(* IEC 61131-3 sources: AXOpen/src/showcase/app/src/components.dukane.welders/Documentation, 3 files *)

(* ---- Axo_IQ_SeriesWelder_Showcase.st ---- *)
USING AXOpen.Core;
NAMESPACE AXOpen.Components.Dukane.Welders
    {S7.extern=ReadWrite}
    CLASS Axo_IQ_SeriesWelder_Showcase EXTENDS AXOpen.Core.AxoObject
        //<ComponentDeclaration>
        VAR PUBLIC
            Dukane_IQ_SeriesWelder : AXOpen.Components.Dukane.Welders.Axo_IQ_SeriesWelder;
        END_VAR
        //</ComponentDeclaration>

        //<InitializationArgumentsDeclaration>
        VAR PUBLIC
            {#ix-set:AttributeName = "<#Activate manual control#>"}
            ActivateManualControl : BOOL;
        END_VAR
        //</InitializationArgumentsDeclaration>

        METHOD PUBLIC OVERRIDE Run
            VAR_INPUT
                inParent : IAxoObject;
            END_VAR

            SUPER.Run(inParent);

            IF ActivateManualControl THEN
                Dukane_IQ_SeriesWelder.ActivateManualControl();
            END_IF;

            //<Initialization>
            Dukane_IQ_SeriesWelder.Run(inParent := THIS, hwID := AXOpen.Showcase.HwIdentifiers#dukaneiqauto_HwID);
            //</Initialization>

        THIS.UseInSequencer();
        END_METHOD

        //<Usage>
        VAR PUBLIC
            {#ix-set:AttributeName = "<#Run test sequence#>"}
            Sequencer   :   AxoSequencer;
            Steps       :   ARRAY[0..12] OF AXOpen.Core.AxoStep;
            Good_Part   :   BOOL;
            Bad_Part    :   BOOL;
            WeldTime    :   DINT;
            WeldEnergy  :   DINT;
            WeldPower   :   DINT;
        END_VAR

        METHOD PRIVATE UseInSequencer
            IF Sequencer.GetContext().OpenCycleCount() = ULINT#0 THEN
                Sequencer.SequenceMode := eAxoSequenceMode#RunOnce;
            END_IF;

            Sequencer.Run(THIS);
            Sequencer.Open();

            IF(Steps[0].Execute(Sequencer, 'Restore')) THEN
                ActivateManualControl := FALSE;
                Dukane_IQ_SeriesWelder.Config.InfoTime    := LTIME#5S;
                Dukane_IQ_SeriesWelder.Config.ErrorTime   := LTIME#10S;
                Dukane_IQ_SeriesWelder.Config.TaskTimeout := LTIME#50S;
                Dukane_IQ_SeriesWelder.Restore();
                Sequencer.MoveNext();
            END_IF;

            IF(Steps[1].Execute(Sequencer, 'ClearError')) THEN
                IF(Dukane_IQ_SeriesWelder.ClearError().IsDone()) THEN
                    Sequencer.MoveNext();
                END_IF;
            END_IF;

            IF(Steps[2].Execute(Sequencer, 'Change welding setup')) THEN
                IF(Dukane_IQ_SeriesWelder.ChangeWeldingSetup(SetupNumber := UINT#2).IsDone()) THEN
                    Sequencer.MoveNext();
                END_IF;
            END_IF;

            IF(Steps[3].Execute(Sequencer, 'Change welding probe')) THEN
                IF(Dukane_IQ_SeriesWelder.ChangeWeldingProbe(ProbeNumber := UINT#1).IsDone()) THEN
                    Sequencer.MoveNext();
                END_IF;
            END_IF;

            IF(Steps[4].Execute(Sequencer, 'RunWeldingWithTime: Setup 2, Probe 1, Time 2s')) THEN
                IF(Dukane_IQ_SeriesWelder.RunWeldingWithTime(SetupNumber := UINT#2, ProbeNumber := UINT#1, WeldingTime := T#2S).IsDone()) THEN
                    Sequencer.MoveNext();
                END_IF;
            END_IF;

            IF(Steps[5].Execute(Sequencer, 'Evaluation OK/NOK')) THEN
                Good_Part   := Dukane_IQ_SeriesWelder.Inputs.SystemStatus.Good_Part;
                Bad_Part    := Dukane_IQ_SeriesWelder.Inputs.SystemStatus.Bad_Part;
                Sequencer.MoveNext();
            END_IF;

            IF(Steps[6].Execute(Sequencer, 'Store results')) THEN
                WeldTime    :=  Dukane_IQ_SeriesWelder.Inputs.CycleWeldTime;
                WeldEnergy  :=  Dukane_IQ_SeriesWelder.Inputs.CycleWeldEnergy;
                WeldPower   :=  Dukane_IQ_SeriesWelder.Inputs.CycleWeldPeakPower;
                Sequencer.MoveNext();
            END_IF;

            IF(Steps[7].Execute(Sequencer, 'Cycle stop')) THEN
                IF(Dukane_IQ_SeriesWelder.CycleStop().IsDone()) THEN
                    Sequencer.MoveNext();
                END_IF;
            END_IF;

            IF(Steps[8].Execute(Sequencer, 'Restore')) THEN
                Dukane_IQ_SeriesWelder.Restore();
                Sequencer.CompleteSequence();
            END_IF;

        END_METHOD

        //</Usage>
    END_CLASS
END_NAMESPACE

(* ---- Axo_IQ_SeriesWelder_Showcase2.st ---- *)
USING AXOpen.Core;
NAMESPACE AXOpen.Components.Dukane.Welders
    {S7.extern=ReadWrite}
    CLASS Axo_IQ_SeriesWelder_Showcase2 EXTENDS AXOpen.Core.AxoObject
        //<ComponentDeclaration>
        VAR PUBLIC
            Dukane_IQ_SeriesWelder : AXOpen.Components.Dukane.Welders.Axo_IQ_SeriesWelder;
        END_VAR
        //</ComponentDeclaration>

        //<InitializationArgumentsDeclaration>
        VAR PUBLIC
            {#ix-set:AttributeName = "<#Activate manual control#>"}
            ActivateManualControl : BOOL;
        END_VAR
        //</InitializationArgumentsDeclaration>

        METHOD PUBLIC OVERRIDE Run
            VAR_INPUT
                inParent : IAxoObject;
            END_VAR

            SUPER.Run(inParent);

            IF ActivateManualControl THEN
                Dukane_IQ_SeriesWelder.ActivateManualControl();
            END_IF;

            //<Initialization>
            Dukane_IQ_SeriesWelder.Run(inParent  :=   THIS,hwID    :=   UINT#60);
            //</Initialization>

        THIS.UseInSequencer();
        END_METHOD

        //<Usage>
        VAR PUBLIC
            Sequencer : AxoSequencer;
            Steps : ARRAY[0..30] OF AXOpen.Core.AxoStep;
        END_VAR

        METHOD PRIVATE UseInSequencer
            IF Sequencer.GetContext().OpenCycleCount() = ULINT#0 THEN
                Sequencer.SequenceMode := eAxoSequenceMode#RunOnce;
            END_IF;

            Sequencer.Run(THIS);
            Sequencer.Open();

            // IF(Steps[0].Execute(Sequencer, 'TemplateMethod_10steps_1')) THEN
            //     IF(Dukane_IQ_SeriesWelder.TemplateMethod_10steps_1().IsDone()) THEN
            //         Sequencer.MoveNext();
            //     END_IF;
            // END_IF;

            // IF(Steps[1].Execute(Sequencer, 'TemplateMethod_10steps_2')) THEN
            //     IF(Dukane_IQ_SeriesWelder.TemplateMethod_10steps_2().IsDone()) THEN
            //         Sequencer.MoveNext();
            //     END_IF;
            // END_IF;

            // IF(Steps[2].Execute(Sequencer, 'TemplateMethod_10steps_3')) THEN
            //     IF(Dukane_IQ_SeriesWelder.TemplateMethod_10steps_3().IsDone()) THEN
            //         Sequencer.MoveNext();
            //     END_IF;
            // END_IF;

            // IF(Steps[3].Execute(Sequencer, 'TemplateMethod_10steps_4')) THEN
            //     IF(Dukane_IQ_SeriesWelder.TemplateMethod_10steps_4().IsDone()) THEN
            //         Sequencer.MoveNext();
            //     END_IF;
            // END_IF;

            // IF(Steps[4].Execute(Sequencer, 'TemplateMethod_10steps_5')) THEN
            //     IF(Dukane_IQ_SeriesWelder.TemplateMethod_10steps_5().IsDone()) THEN
            //         Sequencer.MoveNext();
            //     END_IF;
            // END_IF;

            // IF(Steps[5].Execute(Sequencer, 'TemplateMethod_10steps_6')) THEN
            //     IF(Dukane_IQ_SeriesWelder.TemplateMethod_10steps_6().IsDone()) THEN
            //         Sequencer.MoveNext();
            //     END_IF;
            // END_IF;

            // IF(Steps[6].Execute(Sequencer, 'TemplateMethod_20steps_1')) THEN
            //     IF(Dukane_IQ_SeriesWelder.TemplateMethod_20steps_1().IsDone()) THEN
            //         Sequencer.MoveNext();
            //     END_IF;
            // END_IF;

            // IF(Steps[7].Execute(Sequencer, 'TemplateMethod_20steps_2')) THEN
            //     IF(Dukane_IQ_SeriesWelder.TemplateMethod_20steps_2().IsDone()) THEN
            //         Sequencer.MoveNext();
            //     END_IF;
            // END_IF;

            // IF(Steps[8].Execute(Sequencer, 'TemplateMethod_20steps_3')) THEN
            //     IF(Dukane_IQ_SeriesWelder.TemplateMethod_20steps_3().IsDone()) THEN
            //         Sequencer.MoveNext();
            //     END_IF;
            // END_IF;

            // IF(Steps[9].Execute(Sequencer, 'TemplateMethod_20steps_4')) THEN
            //     IF(Dukane_IQ_SeriesWelder.TemplateMethod_20steps_4().IsDone()) THEN
            //         Sequencer.MoveNext();
            //     END_IF;
            // END_IF;

            // IF(Steps[10].Execute(Sequencer, 'TemplateMethod_20steps_5')) THEN
            //     IF(Dukane_IQ_SeriesWelder.TemplateMethod_20steps_5().IsDone()) THEN
            //         Sequencer.MoveNext();
            //     END_IF;
            // END_IF;

            // IF(Steps[11].Execute(Sequencer, 'TemplateMethod_20steps_6')) THEN
            //     IF(Dukane_IQ_SeriesWelder.TemplateMethod_20steps_6().IsDone()) THEN
            //         Sequencer.MoveNext();
            //     END_IF;
            // END_IF;

            // IF(Steps[12].Execute(Sequencer, 'Restore')) THEN
            //     Dukane_IQ_SeriesWelder.Restore();
            //     Sequencer.CompleteSequence();
            // END_IF;

        END_METHOD

        //</Usage>
    END_CLASS
END_NAMESPACE

(* ---- DukaneWelders.st ---- *)
NAMESPACE AXOpen.Components.Dukane.Welders
    {S7.extern=ReadWrite}
    CLASS DukaneWelders EXTENDS AXOpen.Core.AxoObject
        VAR PUBLIC
            rootObject      : AxoObject;
            axo_IQ_SeriesWelder : AXOpen.Components.Dukane.Welders.Axo_IQ_SeriesWelder_Showcase;
            axo_IQ_SeriesWelder_2 : AXOpen.Components.Dukane.Welders.Axo_IQ_SeriesWelder_Showcase2;
        END_VAR

        METHOD PUBLIC Execute
            rootObject.Run(THIS);
            axo_IQ_SeriesWelder.Run(rootObject);
            axo_IQ_SeriesWelder_2.Run(rootObject);
        END_METHOD
    END_CLASS
END_NAMESPACE
